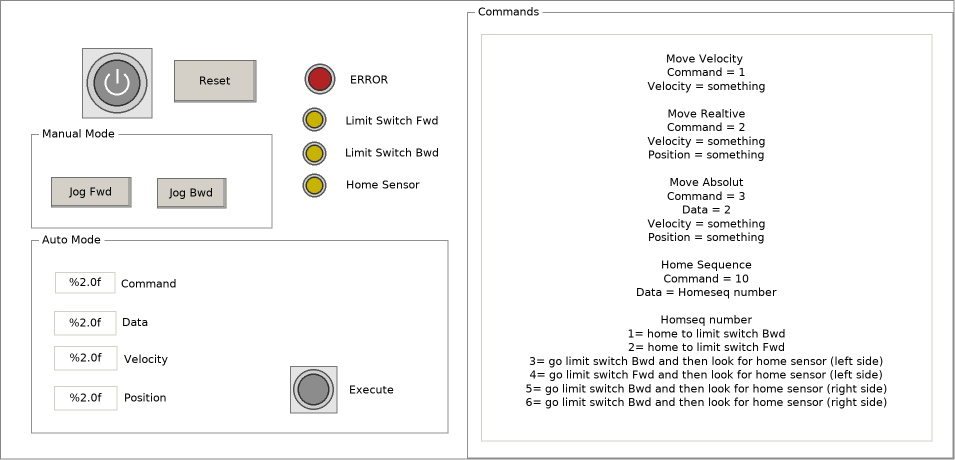
VISUALIZATION FbDriveVisual  // 955x460
    PowerSwitch (82,48 70x70), variable: MAIN.M1.bEnable, behaviour: TOGGLE, style: Switch-PowerSwitch-Gray
    Button (174,60 82x42), "Reset"
        tap MAIN.M1.bReset
    Lamp1 (296,61 48x36), variable: MAIN.M1.bError, style: Lamp-Lamp1-Red
    Label (294,65 150x30), "ERROR"
    GroupBox (31,232 417x201), "Auto Mode"
        Textfield (23,79 62x24), "%2.0f", text variable: MAIN.M1.nCmdData
            OnMouseClick: write MAIN.M1.nCmdData via Default
        Textfield (23,114 63x24), "%2.0f", text variable: MAIN.M1.fVelocity
            OnMouseClick: write MAIN.M1.fVelocity via Default
        Textfield (23,154 63x24), "%2.0f", text variable: MAIN.M1.fPosition
            OnMouseClick: write MAIN.M1.fPosition via Default
        PushSwitch (259,134 47x47), variable: MAIN.M1.bExecute, behaviour: TOGGLE, style: Switch-PushSwitch-Gray
        Label (295,143 91x30), "Execute"
        Label (88,74 75x33), "Data"
        Label (90,111 75x33), "Velocity"
        Label (87,36 74x32), "Command"
        Label (90,150 74x32), "Position"
    Textfield (55,272 60x21), "%2.0f", text variable: MAIN.M1.nCommand
        OnMouseClick: write MAIN.M1.nCommand via Default
    GroupBox (467,4 486x454), "Commands"
        Textfield (14,30 451x407), "Move Velocity Command = 1 Velocity = something Move Realtive Command = 2 Velocity = something Position = something Move Absolut Command = 3 Data = 2 Velocity = something Position = something Home Sequence Command = 10 Data = Homeseq number Homseq number 1= home to limit switch Bwd 2= home to limit switch Fwd 3= go limit switch Bwd and then look for home sensor (left side) 4= go limit switch Fwd and then look for home sensor (left side) 5= go limit switch Bwd and then look for home sensor (right side) 6= go limit switch Bwd and then look for home sensor (right side)"
    Label (317,106 150x30), "Limit Switch Fwd"
    Label (317,138 150x30), "Limit Switch Bwd"
    Label (308,170 150x30), "Home Sensor"
    Lamp1 (301,106 27x27), variable: not MAIN.M1.bLimitFwd, style: Lamp-Lamp1-Yellow
    Lamp1 (301,140 27x27), variable: not MAIN.M1.bLimitBwd, style: Lamp-Lamp1-Yellow
    Lamp1 (301,172 27x27), variable: MAIN.M1.bHomeSensor, style: Lamp-Lamp1-Yellow
    GroupBox (31,126 241x102), "Manual Mode"
        Button (126,52 69x30), "Jog Bwd"
            tap MAIN.M1.bJogBwd
        Button (20,51 80x30), "Jog Fwd"
            tap MAIN.M1.bJogFwd
END_VISUALIZATION

(* stored: Version 1.1.0.1, ProductVersion 3.1.4022.10
   Visu FbDriveVisual: Id {eec707a1-ae81-4ed5-b43d-3a6c88c2ea88} *)
